SYSTEM MapToCommandTest
  (* Version 1.0, 2026-02-23, 4diac test *)
  APPLICATION App
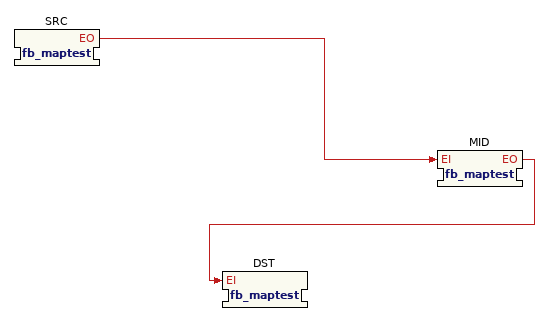
    FBS
      SRC : fb_maptest;
      MID : fb_maptest;
      DST : fb_maptest;
    END_FBS
    EVENT_CONNECTIONS
      SRC.EO TO MID.EI;
      MID.EO TO DST.EI;
    END_CONNECTIONS
  END_APPLICATION
  DEVICE Device1 : TEST_DEVICE(MGR_ID := "localhost:61499" (* Device manager socket ID *))
    RESOURCE Res1 : TEST_RES
    END_RESOURCE
  END_DEVICE
  MAPPINGS
    App.SRC ON Device1.Res1;
    App.DST ON Device1.Res1;
  END_MAPPINGS
END_SYSTEM
